Universal Robots PolyScope program: 3exMath.urp

Program 3exMath (installation=default directory=/home/ur/ursim-current/programs createdIn=5.11.8.1010444 lastSavedIn=5.11.8.1010444 robotSerialNumber=20195399999)
Calibrated DH parameters: a=[0, -0.24355, -0.2132, 0, 0, 0]; d=[0.15185, 0, 0, 0.13105, 0.08535, 0.0921]; alpha=[1.570796, 0, 0, 1.570796, -1.570796, 0]; deltaTheta=[0, 0, 0, 0, 0, 0]
BeforeStart
  Script file /home/ur/ursim-current/programs/Script/3_Ex_Math.script
    | def Calc(a, b):
    | 	c = a + b
    | 	global d = a - b
    | 	return c
    | end
Robot Program (runOnlyOnce=false)
  Wait Sleep waitTime=0.01
  var_1 := a
  var_2 := b
  Script: Result=Calc(var_1, var_2)
  var_3 := Result
  var_4 := d
